FUNCTION_BLOCK FB_Sensor
VAR_INPUT
	bSensorSignal: BOOL;
	bRequestedState: BOOL;
	bCheckState: BOOL;
	uiErrorOnDelay_MS: UINT:=1000;
	uiSensorOnDelay_MS: UINT:=100;
	uiErrorOffDelay_MS: UINT:=1000;
	uiSensorOffDelay_MS: UINT:=100;
	bSimulationON: BOOL;
	
END_VAR
VAR_OUTPUT
END_VAR
VAR
	fbSensorON_TON :TON;
	fbSensorOFF_TON :TON;
	fbSensorErrorON_TON:TON;
	fbSensorErrorOFF_TON:TON;
END_VAR

IF bSimulationON THEN
	bSensorSignal:=bRequestedState;
END_IF
fbSensorON_TON(IN:=bSensorSignal AND bRequestedState, PT:=UINT_TO_TIME(uiSensorOnDelay_MS));
fbSensorOFF_TON(IN:=NOT bSensorSignal AND NOT bRequestedState, PT:=UINT_TO_TIME(uiSensorOffDelay_MS));
fbSensorErrorON_TON(IN:=NOT bSensorSignal AND bRequestedState AND bCheckState, PT:=UINT_TO_TIME(uiErrorOnDelay_MS));
fbSensorErrorOFF_TON(IN:=bSensorSignal AND NOT bRequestedState AND bCheckState, PT:=UINT_TO_TIME(uiErrorOffDelay_MS));

bCheckState:= FALSE;

{attribute 'monitoring':= 'call'}
PROPERTY prSensorOffError : BOOL
GET
prSensorOffError := fbSensorErrorON_TON.Q;
END_GET
END_PROPERTY

{attribute 'monitoring':= 'call'}
PROPERTY prSensorOffOK : BOOL
GET
prSensorOffOK := fbSensorOFF_TON.Q;
END_GET
END_PROPERTY

{attribute 'monitoring':= 'call'}
PROPERTY prSensorOnError : BOOL
GET
prSensorOnError := fbSensorErrorOFF_TON.Q;
END_GET
END_PROPERTY

{attribute 'monitoring':= 'call'}
PROPERTY prSensorOnOK : BOOL
GET
prSensorOnOK := fbSensorON_TON.Q;
END_GET
END_PROPERTY

END_FUNCTION_BLOCK

(* stored: Version 1.1.0.1, ProductVersion 3.1.4024.15
   POU FB_Sensor: Id {b3b43494-dfbd-47ae-9555-8a34c9c3c813}, SpecialFunc None
   Property prSensorOffError: Id {dd4317be-7bc1-4d2a-8186-9301df986d98}
   Get Get: Id {3580e491-1f8e-43f1-881f-9227f1824b8c}
   Property prSensorOffOK: Id {2b0882da-dd02-45d0-8fe7-88a9145a68c4}
   Get Get: Id {02430664-efde-45b0-bd8b-821e27c8019a}
   Property prSensorOnError: Id {eb28fc78-11a4-414b-8d7f-148280868fb0}
   Get Get: Id {b0149dda-ac15-4bb9-9159-06882874d057}
   Property prSensorOnOK: Id {d2e1803d-eab4-47e0-8e03-607f7dc9e6b1}
   Get Get: Id {7eb509e8-e5a7-4018-a468-a7f7fd331266} *)
